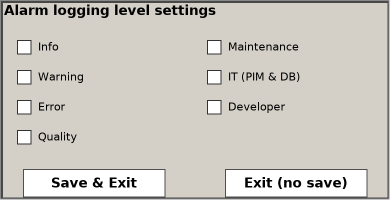
VISUALIZATION vAlarmLogSetup_Dialog  // 390x200
VAR_IN_OUT
	uiAllarmLogSettings:UINT;
END_VAR
    Rectangle (1,1 388x198), "Alarm logging level settings"
    Rectangle (23,169 142x28), "Save & Exit"
        OnMouseClick: CloseDialog Dialog=vAlarmLogSetup_Dialog, Result=OK, NumpadKeypadSet=True
    Rectangle (225,169 142x28), "Exit (no save)"
        OnMouseClick: CloseDialog Dialog=vAlarmLogSetup_Dialog, Result=Cancel, NumpadKeypadSet=True
    Checkbox (15,32 175x30), "Info", variable: uiAllarmLogSettings.0
    Checkbox (15,62 175x30), "Warning", variable: uiAllarmLogSettings.1
    Checkbox (15,92 175x30), "Error", variable: uiAllarmLogSettings.2
    Checkbox (15,122 175x30), "Quality", variable: uiAllarmLogSettings.3
    Checkbox (205,32 175x30), "Maintenance", variable: uiAllarmLogSettings.4
    Checkbox (205,62 175x30), "IT (PIM & DB)", variable: uiAllarmLogSettings.5
    Checkbox (205,92 175x30), "Developer", variable: uiAllarmLogSettings.6
END_VISUALIZATION

(* stored: Version 1.1.0.1, ProductVersion 3.1.4024.12
   Visu vAlarmLogSetup_Dialog: Id {577041a2-a19c-476a-a22d-be62fcc74663} *)
